// TIA Portal V16 export
// export: Created 2021-03-04T22:03:59.602254Z, ExportSetting WithDefaults, DisplayName Totally Integrated Automation Portal, DisplayVersion V16, DisplayName TIA Portal Version Control Interface, DisplayVersion V16, DisplayName TIA Portal Openness, DisplayVersion V16, DisplayName SINAMICS Startdrive Advanced, DisplayVersion V16, DisplayName SINAMICS Startdrive G130, G150, S120, S150, SINAMICS MV, S210, DisplayVersion V16, DisplayName SINAMICS Startdrive G110M, G120, G120C, G120D, G120P, DisplayVersion V16, DisplayName STEP 7 Professional, DisplayVersion V16, DisplayName STEP 7 Safety, DisplayVersion V16, DisplayName WinCC Professional, DisplayVersion V16
FUNCTION_BLOCK "fbRackLights"   // FB6, LAD
{ S7_Optimized_Access := 'TRUE' }
VERSION : 0.1
// stored: AutoNumber true, IsIECCheckEnabled false, IsRetainMemResEnabled false, MemoryReserve 100, SetENOAutomatically false, UDAEnableTagReadback false
   VAR_INPUT
      iInDelaySecs { ExternalAccessible := 'False'; ExternalVisible := 'False'; ExternalWritable := 'False'} : Int;
      rInCurrentTemperature : Real;
   END_VAR
   VAR_OUTPUT
      bOutLights { ExternalAccessible := 'False'; ExternalVisible := 'False'; ExternalWritable := 'False'} : Bool;
   END_VAR
   VAR RETAIN
      Controls { ExternalVisible := 'False'} : Struct
         iMode { ExternalVisible := 'False'} : Int;   // 0: Off, 1: On, 2: Auto
         diOffTime { ExternalVisible := 'False'} : DInt;   // Off time (seconds past midnight)
         diOnTime { ExternalVisible := 'False'} : DInt;   // On time (seconds past midnight)
         rHighTemperatureLimit { ExternalVisible := 'False'} : Real := 75.0;
      END_STRUCT;
      Status { ExternalVisible := 'False'; ExternalWritable := 'False'} : Struct
         diSecondsElapsed { ExternalVisible := 'False'; ExternalWritable := 'False'} : DInt;
      END_STRUCT;
   END_VAR
   VAR
      bLightsCommand { ExternalAccessible := 'False'; ExternalVisible := 'False'; ExternalWritable := 'False'} : Bool;
   END_VAR
   VAR RETAIN
      TON_OnDelay { ExternalAccessible := 'False'; ExternalVisible := 'False'; ExternalWritable := 'False'; S7_SetPoint := 'True'} : TON_TIME;
   END_VAR
   VAR_TEMP
      tCurrentDateTime : Date_And_Time;   // Current PLC Date and Time
      tCurrentTimeMilli : Time_Of_Day;   // Current time (ms since 0:00:00)
      retVal : Int;   // Garbage return value from RD_LOC_T
      diSeconds : DInt;
   END_VAR
   VAR CONSTANT
      eOffMode : Int := 0;
      eOnMode : Int := 1;
      eAutoMode : Int := 2;
   END_VAR
BEGIN

REGION Network 1 (SCL): State 0 - Off Mode and State 1 - On Mode
   // Directly assign rack light output based on off or on mode
   IF #Controls.iMode = #eOffMode THEN
       #bLightsCommand := 0;
   ELSIF #Controls.iMode = #eOnMode THEN
       #bLightsCommand := 1;
   END_IF;
END_REGION

REGION Network 2 (SCL): State 2 - Auto Mode
   // Check the current time against the on time and off time, and assign the lights appropriately
   IF #Controls.iMode = #eAutoMode THEN

       //Get current time from PLC and convert to seconds since 0:00:00
       #retVal := RD_LOC_T(OUT => #tCurrentDateTime);
       #tCurrentTimeMilli := DT_TO_TOD(IN := #tCurrentDateTime);
       #diSeconds := TOD_TO_DINT(IN := #tCurrentTimeMilli)/1000; //Go from ms time to DInt seconds

       // Situation 1: Off time happens after on time
       IF #Controls.diOffTime > #Controls.diOnTime THEN 
           IF #diSeconds > #Controls.diOnTime AND #diSeconds < #Controls.diOffTime THEN
               #bLightsCommand := 1;
           ELSE
               #bLightsCommand := 0;
           END_IF;

       // Situation 2: On time happens after off time
       ELSE
           IF #diSeconds > #Controls.diOffTime AND #diSeconds < #Controls.diOnTime THEN
               #bLightsCommand := 0;
           ELSE
               #bLightsCommand := 1;
           END_IF;
       END_IF;
   END_IF;
END_REGION

REGION Network 3 (SCL): Temperature Override When in Auto

   IF #Controls.iMode = #eAutoMode AND #rInCurrentTemperature > #Controls.rHighTemperatureLimit THEN
       #bLightsCommand := 0;
   END_IF;
END_REGION

REGION Network 4 (SCL): Write seconds elapsed status and set outputs with confugred delay
   #Status.diSecondsElapsed := #diSeconds;

   #TON_OnDelay(IN := #bLightsCommand,
                PT := INT_TO_TIME(#iInDelaySecs));

   #bOutLights := #TON_OnDelay.Q;
END_REGION
END_FUNCTION_BLOCK
